(* CODESYS project ScaraTrackingFinal（运动控制2）.project

Project tree, tasks and I/O mapping:
  Device : CODESYS Softmotion RTE V3 x64_test, 3S - Smart Software Solutions GmbH, order no. 001, version 3.5.15.20
    application Application
      libraries: Standard, * (System); VisuDialogs, * (System)
      task MainTask (cyclic, interval t#20ms, priority 1) calls MainPRG
      task VISU_TASK (cyclic, interval 100 ms, priority 31) calls VisuElems.Visu_Prg
      task SoftMotion_PlanningTask (freewheeling, priority 15) calls SoftMotion_PlanningPrg
      axis group MyScara: TRAFO.Kin_Scara2_Z, axes DriveA, DriveB, DriveZ
      visualisation TargetVisuStart
      Depictor
      function block FB_PositionIterator2 [ST]
      trace Trace (task MainTask): PLC_PRG.RAP.Position.c.X, PLC_PRG.RAP.Position.c.Y, PLC_PRG.RAV.Velocity.c.X, PLC_PRG.RAV.Velocity.c.Y
      program MainPRG [SFC]: EnableDrives_active, SetMCS_active, SetMCS_exit, SetTable_active, DoMove_active
      program SoftMotion_PlanningPrg [ST]
    SoftMotion General Axis Pool
      DriveA : SM_Drive_Virtual, 3S - Smart Software Solutions GmbH, order no. 1805, version 4.0.0.0
          settings: wDriveID = 9; fSWMaxVelocity = 400; fSWLimitPositive = 190; fSWLimitNegative = -190
      DriveB : SM_Drive_Virtual, 3S - Smart Software Solutions GmbH, order no. 1805, version 4.0.0.0
          settings: wDriveID = 10; fSWMaxVelocity = 400; fSWLimitPositive = 135; fSWLimitNegative = -135
      DriveZ : SM_Drive_Virtual, 3S - Smart Software Solutions GmbH, order no. 1805, version 4.0.0.0
          settings: wDriveID = 11; fSWMaxVelocity = 400
      RotaryTable : SM_Drive_Virtual, 3S - Smart Software Solutions GmbH, order no. 1805, version 4.0.0.0
          settings: wDriveID = 12; iMovementType = 0; fSWMaxVelocity = 100
  libraries: DepictorBase, 1.0.4.0 (3S - Smart Software Solutions GmbH)
  text list GlobalTextList
*)

// Device/Application/MainPRG
PROGRAM MainPRG
VAR
	MC_TrackRotaryTable_0: MC_TrackRotaryTable;
    
	MC_MoveDirectAbsolute_0: MC_MoveDirectAbsolute;
	MC_GroupEnable_0: MC_GroupEnable;
	FB_PositionIterator_0: FB_PositionIterator2;
	MC_Power_A: MC_Power;
    MC_Power_B: MC_Power;
	MC_Power_Z: MC_Power;
	MC_Power_RT: MC_Power;
	_Done: BOOL;
	MC_SetCoordinateTransform_0: MC_SetCoordinateTransform;
	OffsetMCS_WCS: SM3_Robotics.MC_COORD_REF := (Z := 400);
	MC_Jog_0: MC_Jog := (Velocity := 50, Acceleration := 100, Deceleration := 100);
    OffsetRT_WCS: SM3_Robotics.MC_COORD_REF := (X := 400, Y := 600);
    OffsetPCS_RT: SM3_Robotics.MC_COORD_REF := (X := 200, Y := 200, Z := 10, A := 45);
END_VAR
VAR // added by the converter: edge detectors and wires of the graphical bodies
    _w1 : BOOL;
END_VAR

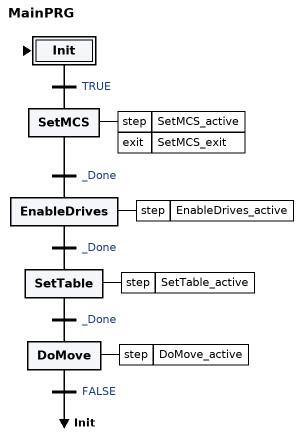
INITIAL_STEP Init:
END_STEP
TRANSITION FROM Init TO SetMCS
    := TRUE;
END_TRANSITION
STEP SetMCS:
    SetMCS_active(N);  // step action
    SetMCS_exit(P0);  // exit action
END_STEP
TRANSITION FROM SetMCS TO EnableDrives
    := _Done;
END_TRANSITION
STEP EnableDrives:
    EnableDrives_active(N);  // step action
END_STEP
TRANSITION FROM EnableDrives TO SetTable
    := _Done;
END_TRANSITION
STEP SetTable:
    SetTable_active(N);  // step action
END_STEP
TRANSITION FROM SetTable TO DoMove
    := _Done;
END_TRANSITION
STEP DoMove:
    DoMove_active(N);  // step action
END_STEP
TRANSITION FROM DoMove TO Init
    := FALSE;
END_TRANSITION

ACTION EnableDrives_active:
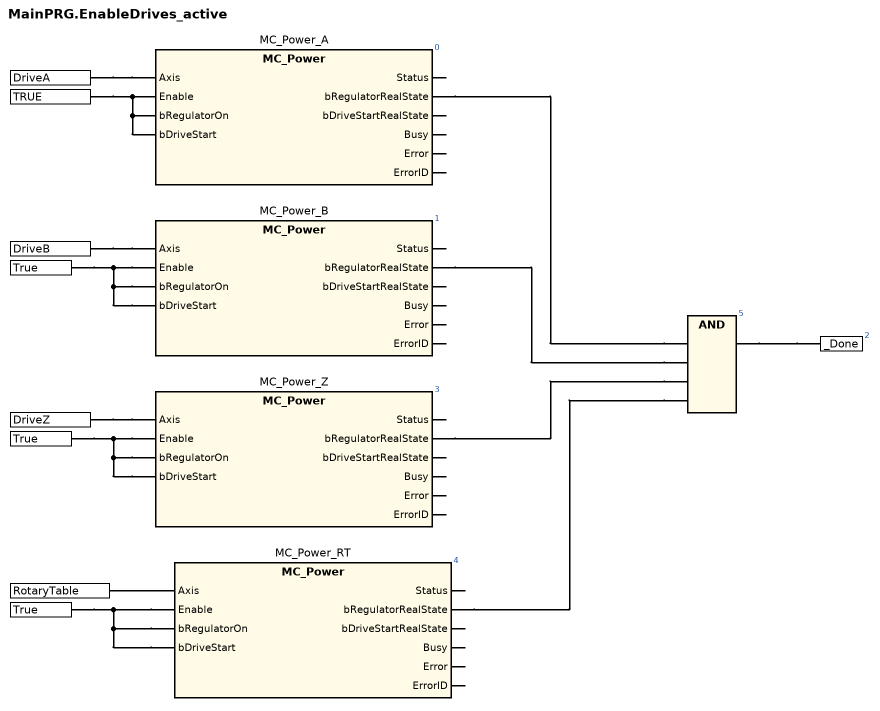
MC_Power_A(Axis := DriveA, Enable := TRUE, bRegulatorOn := TRUE, bDriveStart := TRUE); // MC_Power
MC_Power_B(Axis := DriveB, Enable := True, bRegulatorOn := True, bDriveStart := True); // MC_Power
_Done := _w1;
MC_Power_Z(Axis := DriveZ, Enable := True, bRegulatorOn := True, bDriveStart := True); // MC_Power
MC_Power_RT(Axis := RotaryTable, Enable := True, bRegulatorOn := True, bDriveStart := True); // MC_Power
_w1 := MC_Power_A.bRegulatorRealState AND MC_Power_B.bRegulatorRealState AND MC_Power_Z.bRegulatorRealState AND MC_Power_RT.bRegulatorRealState;
END_ACTION

ACTION SetMCS_active:
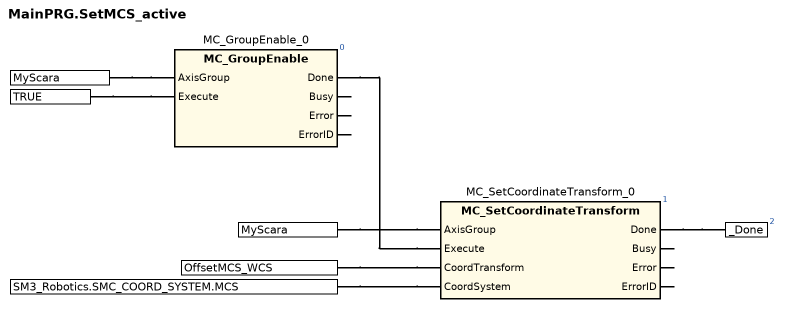
MC_GroupEnable_0(AxisGroup := MyScara, Execute := TRUE); // MC_GroupEnable
MC_SetCoordinateTransform_0(
    AxisGroup := MyScara,
    Execute := MC_GroupEnable_0.Done,
    CoordTransform := OffsetMCS_WCS,
    CoordSystem := SM3_Robotics.SMC_COORD_SYSTEM.MCS); // MC_SetCoordinateTransform
_Done := MC_SetCoordinateTransform_0.Done;
END_ACTION

ACTION SetMCS_exit:
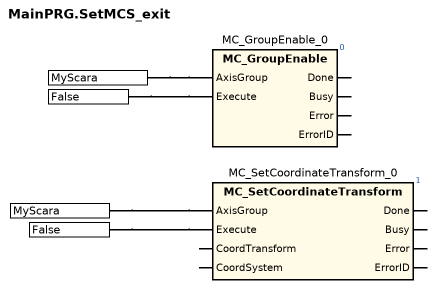
MC_GroupEnable_0(AxisGroup := MyScara, Execute := False); // MC_GroupEnable
MC_SetCoordinateTransform_0(AxisGroup := MyScara, Execute := False); // MC_SetCoordinateTransform
END_ACTION

ACTION SetTable_active:
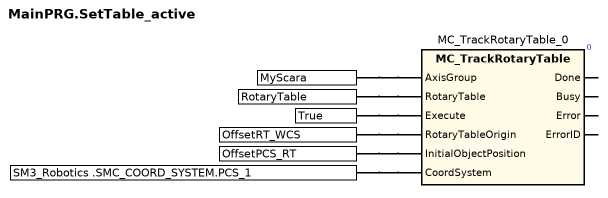
MC_TrackRotaryTable_0(
    AxisGroup := MyScara,
    RotaryTable := RotaryTable,
    Execute := True,
    RotaryTableOrigin := OffsetRT_WCS,
    InitialObjectPosition := OffsetPCS_RT,
    CoordSystem := SM3_Robotics .SMC_COORD_SYSTEM.PCS_1); // MC_TrackRotaryTable
END_ACTION

ACTION DoMove_active:
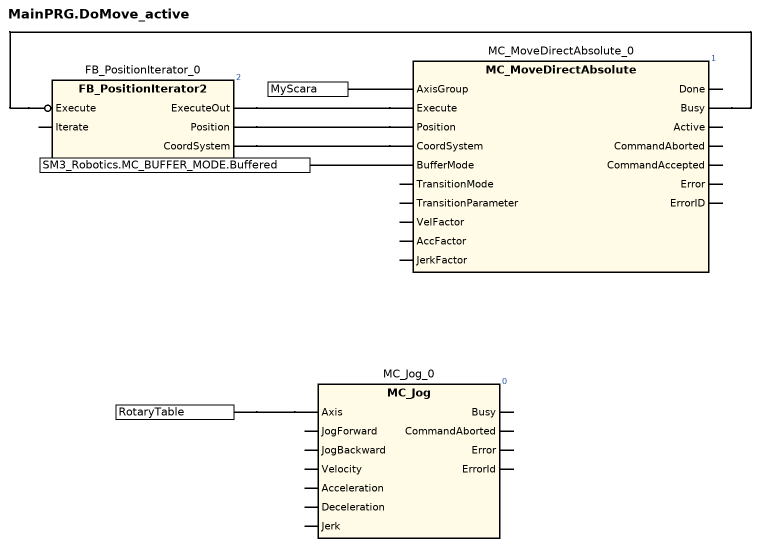
MC_Jog_0(Axis := RotaryTable); // MC_Jog
MC_MoveDirectAbsolute_0(
    AxisGroup := MyScara,
    Execute := FB_PositionIterator_0.ExecuteOut,
    Position := FB_PositionIterator_0.Position,
    CoordSystem := FB_PositionIterator_0.CoordSystem,
    BufferMode := SM3_Robotics.MC_BUFFER_MODE.Buffered); // MC_MoveDirectAbsolute
FB_PositionIterator_0(Execute := NOT MC_MoveDirectAbsolute_0.Busy); // FB_PositionIterator2
END_ACTION

END_PROGRAM

// Device/Application/FB_PositionIterator2
FUNCTION_BLOCK FB_PositionIterator2
VAR_INPUT
    Execute: BOOL;
    Iterate: BOOL;
END_VAR
VAR_OUTPUT
    ExecuteOut: BOOL;
    Position: SM3_Robotics.SMC_POS_REF;
    CoordSystem: SM3_Robotics.SMC_COORD_SYSTEM:= SM3_Robotics.SMC_COORD_SYSTEM.PCS_1;
END_VAR
VAR
	_oldExecute: BOOL;
	_i: DINT:= 0;
    _aPositions: ARRAY [0..3] OF SMC_POS_REF := [(c := (X := -75, Y := -75, Z := 0)), (c := (X := 75, Y := -75, Z := 0)), (c := (X := 75, Y := 75, Z := 0)), (c := (X := -75, Y := 75, Z := 0))];
	_FirstRun: BOOL := TRUE;
END_VAR

IF Execute AND NOT _oldExecute  THEN
    _i := _i + 1;
    IF _i > 3 THEN
        _i := 0;
    END_IF
END_IF
Position:= _aPositions[_i];
ExecuteOut:= Execute AND Iterate OR _FirstRun;
_oldExecute:= Execute;
_FirstRun:= FALSE;

END_FUNCTION_BLOCK

// Device/Application/SoftMotion_PlanningPrg
PROGRAM SoftMotion_PlanningPrg

;

END_PROGRAM

// Device/Application/TargetVisuStart
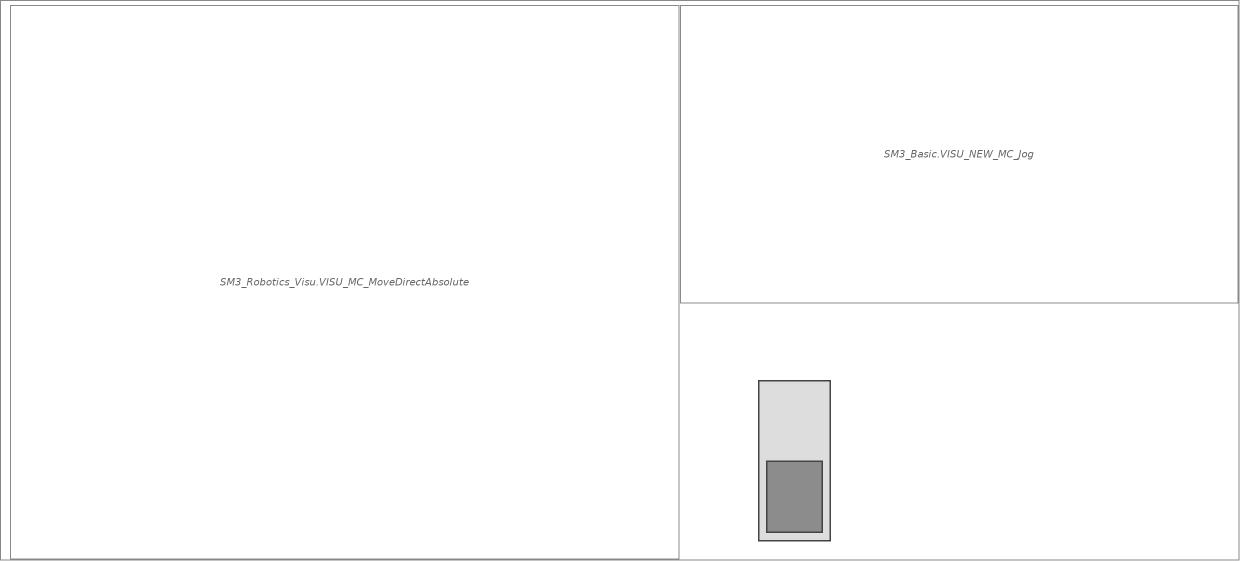
VISUALIZATION TargetVisuStart  // 1240x561
    Frame (10,5 669x554)
        shows SM3_Robotics_Visu.VISU_MC_MoveDirectAbsolute(m_Input_FB := MainPRG.MC_MoveDirectAbsolute_0)
    Frame (680,5 558x298)
        shows SM3_Basic.VISU_NEW_MC_Jog(m_Input_FB := MainPRG.MC_Jog_0)
    DipSwitch (700,380 189x161), variable: MainPRG.FB_PositionIterator_0.Iterate, behaviour: TOGGLE, style: Switch-DipSwitch-Gray
END_VISUALIZATION
